(* IEC 61131-3 sources: SJ_AGV/PLC/Standard_functions.4.4.0/CarrierControl, 6 files *)

(* ---- AutoInsert_FB.ST ---- *)
FUNCTION_BLOCK AutoInsert_FB
VAR_EXTERNAL
	NDC8 : NDC8_T;
	INPUT : INPUT_T;

END_VAR

VAR_INPUT

END_VAR

VAR_OUTPUT
		InProgress : BOOL;
		NotInsideTargetSafety : BOOL;
		Failed : BOOL;

END_VAR

VAR

END_VAR
(*************************************************************************************
 		Automatic insert of vehicle into system
**************************************************************************************)

(**************************************************************************************)
(* Make readable/understandable signals

	OUTPUTS	*)
InProgress				:= (NDC8.Autoinsert.Target>0) and not NDC8.LayoutPosition.InSystem;
NotInsideTargetSafety 	:= InProgress and not NDC8.Autoinsert.OnSegment;
Failed					:= (InProgress and NDC8.Guidance.OutsideSafetyZone)
														   or
														   (
																NDC8.Opt.VehicleStatusID = 5
																or NDC8.Opt.VehicleStatusID = 11
														   );

case NDC8.VehicleControl.OperationMode of
	0: 												(* In automatic mode 							*)
		if INPUT.Reset_PB then		(* if reset button pressed 						*)
			NDC8.Manual.PlcSpeed := 50;			(* Set autoinsert speed to 100mm/s 				*)
		else
			NDC8.Manual.PlcSpeed := 0;
		end_if;

	2:
		if ndc8.mcd.Button4 and ndc8.mcd.Button5 then	(* forward slow *)
			ndc8.manual.PlcSpeed := 300 ;
		else
			ndc8.manual.PlcSpeed := 0 ;
		end_if;
else
	;												(* Don't override MCD in semi mode. 			*)
end_case;

END_FUNCTION_BLOCK

(* ---- CARRIERCONTROL_FB.ST ---- *)
FUNCTION_BLOCK CARRIERCONTROL_FB
VAR_EXTERNAL
	(** IN **)
	NDC8 : NDC8_T;

END_VAR

VAR_INPUT
	FlexSlowdown,
	LS2000Slowdown	: bool;
END_VAR

VAR_OUTPUT
	AutoInsertNotInsideTargetSafety : bool;
	AutoinsertInProgress			: bool;
	StartDelayStartWarning			: bool;
END_VAR

VAR

	AutoInsert : AutoInsert_FB;
	SlowDown : Slowdown_FB;
	StartDelay : StartDelay_FB;
	EStopFB : EStop_FB;
	ResetButtonFB : ResetButton_FB;

	MasterLink_TOF	: TOF;

	MasterLinkUp_RT,
	BbxDone_RT,
	NDC8LibFail_RT,
	StandardFBFail_RT		: R_Trig;

	MasterLink_FT		: F_Trig;

	to_bytes : NDC8_STRING_TO_BYTES;
	to_dec : ASCII_TO_DEC;
	AccessPointB5,
	AccessPointB6,
	AccessPointB5b1A,
	AccessPointB5b2A,
	AccessPointB6b1A,
	AccessPointB6b2A,
	AccessPointB5b1,
	AccessPointB6b1,
	AccessPointB5b2,
	AccessPointB6b2,
	MasterLink		 : dint;
	NDC8LibFail,
	StandardFBFail : bool;

	BlackboxFB : Blackbox_FB;

END_VAR
(*
------------------------------------------------------------------------------------
 CARRIER_CONTROL_FB
 ------------------

 Description:
 Handles symbols essential for driving the vehicle
 -------------------------------------------------------------------------------------*)

(**************************************************************************************)

AutoInsert();
Slowdown(	FlexSlowdown := FlexSlowdown,
			LS2000Slowdown := LS2000Slowdown); 			(* Slow down vehicle *)
StartDelay();			(* Start delay after estop *)
EStopFB();
ResetButtonFB();

(**************************************************************************************)

(* Version verification  *)

(**************************************************************************************)
(* ALTRENATIVE CREEP DISTANCE  *)
if NDC8.UserDefined.NormalCreepDistance = 0 then
	NDC8.UserDefined.NormalCreepDistance := NDC8.Vehicle.CreepDistance;
end_if;

(**************************************************************************************)
(* Do not allow download from Application Designer while vehicle is moving *)
NDC8.VehicleControl.PreventAppDownload := NDC8.VehicleControl.Moving;

(**************************************************************************************)
(* Events 		 *)

(* Convert Access points MAC adress xx.xx.xx.xx.b1.b2 from ASCII to dint *)

to_bytes(str:= NDC8.Wlan.AccessPoint);					(* Converts string to bytes *)
AccessPointB5b1A := byte_to_dint(to_bytes.bytes[13]);
AccessPointB5b2A := byte_to_dint(to_bytes.bytes[14]);
AccessPointB6b1A := byte_to_dint(to_bytes.bytes[16]);
AccessPointB6b2A := byte_to_dint(to_bytes.bytes[17]);

to_dec(ASCII:= AccessPointB5b1A);						(* Convert from ASCII to decimal *)
AccessPointB5b1  := to_dec.dec;
to_dec(ASCII:= AccessPointB5b2A);
AccessPointB5b2  := to_dec.dec;
to_dec(ASCII:= AccessPointB6b1A);
AccessPointB6b1  := to_dec.dec;
to_dec(ASCII:= AccessPointB6b2A);
AccessPointB6b2  := to_dec.dec;

MasterLink_TOF(IN:=NDC8.Master.MasterLinkUp, PT:=t#10s);(* Connection is down for more than 10 seconds. *)
MasterLink_FT(CLK:= MasterLink_TOF.q); 					(* Only generate event when connection is lost, not during boot. *)
Case MasterLink of
	0: 	if NDC8.Master.MasterLinkUp then
		(* Found connection to system manager. *)
			MasterLink := 10;
		end_if;
	10: if MasterLink_FT.q then									(* Lost connection to system manager. *)
		BbxTrig := (NDC8.VehicleControl.OperationMode=0);		(* Create blackbox if vehicle is in Automatic Mode. *)
		a:=TRACE_bool('BbxTrig',BbxTrig);
		a:=TRACE_string('MasterLink down');
		NDC8.Blackbox.TrigReason:='MasterLink down';
		MasterLink := 0;
	end_if;
end_case;

(**************************************************************************************)
(* Stop while master controller is minimizes the segments allocated, during detouring. TS40 in NDC demo. *)

if NDC8.VehicleControl.HaltRequest and not StopHalt then
    StopHalt:= True;
    NDC8.VehicleControl.HaltRequestDone:=True;
elsif not NDC8.VehicleControl.HaltRequest and StopHalt then
    NDC8.VehicleControl.HaltRequestDone:=False;
    StopHalt:= False;
end_if;

(* G5 CHECK BATTERY OVER VOLTAGE *)

(**************************************************************************************)
(* 			DEBUG handling *)

if BbxTrig then
	BlackboxFB();
end_if;

BbxDone_RT(CLK:=BlackboxFB.finished);
if BbxDone_RT.q then
	BbxTrig := false;
	a:=TRACE_bool('BbxTrig',BbxTrig);
	NDC8.Blackbox.TrigReason:='Default';
end_if;

(**************************************************************************************)
(* 			Outputs *)
AutoinsertInProgress			:= Autoinsert.InProgress;
AutoInsertNotInsideTargetSafety := AutoInsert.NotInsideTargetSafety;
StartDelayStartWarning			:= StartDelay.StartWarning;

END_FUNCTION_BLOCK

(* ---- ESTOP_FB.ST ---- *)
FUNCTION_BLOCK ESTOP_FB
VAR_EXTERNAL
	NDC8 : NDC8_T;
	INPUT : INPUT_T;
END_VAR

VAR_INPUT

END_VAR

VAR_OUTPUT

END_VAR

VAR
	EstopRT		 	: R_trig;
	EstopFT		 	: R_trig;
	EstopPBRT	 	: R_trig;
END_VAR
(**************************************************************************************)
(* E-STOP BUTTONS: *)

StopEstopButton := INPUT.EstopStop_PB and NDC8.VehicleControl.OperationMode <> 1;	(* Estop push button in all modes except manual *)
StopReset		:= StopReset OR StopEstopButton;									(* This stop signal needs to be reset	*)

(* Display Vehicle E-Stopped *)
DisplayStopString(INStatus:=StopEstopButton, StopString:=8, StopValue:=0);

(* Event  Estop pushbutton ON *)
EStopPBRT(CLK:=StopEstopButton);
if EStopPBRT.Q then
	;
end_if;

(* Event  Estop ON * )

EStopRT(CLK:=NDC8.VehicleControl.Estop);
EStopFT(CLK:=NDC8.VehicleControl.Estop);
if EStopRT.Q then
	EventQueue(EventCode:=100,
			Par1:=NDC8.LayoutPosition.Segment,
			Par2:=0,
			Par3:=0,
			Par4:=0);
	a:=TRACE_DINT('EventCode', EventQueue.EventCode);
end_if;
*)

END_FUNCTION_BLOCK

(* ---- RESETBUTTON_FB.ST ---- *)
FUNCTION_BLOCK RESETBUTTON_FB
VAR_EXTERNAL
	NDC8 : NDC8_T;
	INPUT : INPUT_T;

END_VAR

VAR_INPUT

END_VAR

VAR_OUTPUT

END_VAR

VAR
	StopResetRT,
	ResetButtonRT 	 : r_trig;
	EstopFT,
	ResetButtonFT	 : F_Trig;

END_VAR
(**************************************************************************************)
(* RESET STOP: *)
StopResetRT(CLK:=StopReset);
ResetButtonRT(CLK:=Input.Reset_PB);
ResetButtonFT(CLK:=Input.Reset_PB);

(* Reset push needed *)
if ResetButtonRT.Q and NDC8.LayoutPosition.InSystem then 			(* Set stop signal while button is pressed,
																	so the vehicle does not start to drive,
																	except during autoinsert or during override of rear obstacle *)
	StopResetButton := true;
end_if;

if Input.Reset_PB
	or Input.TillerArmDown
	or Input.GateOpen
	or Input.PlatformNotUpperPos then												(* Release StopReset bit when pressing the button *)
		StopReset 	:= false;
end_if;

if ResetButtonFT.Q or
	NDC8.VehicleControl.OperationMode = 1 then
		StopReset 						:= false;
		StopResetButton 				:= false;
end_if;

InStatus	:= 	StopReset and NDC8.VehicleControl.OperationMode <> 0;
DisplayStopString(INStatus:=InStatus, StopString:=74, StopValue:=0);

InStatus	:= 	StopResetButton	and NDC8.VehicleControl.OperationMode <> 0;
DisplayStopString(INStatus:=InStatus, StopString:=124, StopValue:=0);

END_FUNCTION_BLOCK

(* ---- SLOWDOWN_FB.ST ---- *)
FUNCTION_BLOCK SLOWDOWN_FB
VAR_EXTERNAL
	NDC8 : NDC8_T;
	INPUT : INPUT_T;

END_VAR

VAR_INPUT
	FlexSlowdown,
	LS2000Slowdown	: bool;
END_VAR

VAR_OUTPUT

END_VAR

VAR
	CurrentVehicleSpeed : DINT;
	VehicleSlowDownSpeed : DINT;
	SlowDownTOF : TOF;
	SlowDownKeep : BOOL;
END_VAR
(*************************************************************************************
 		SLOW DOWN
**************************************************************************************)
CurrentVehicleSpeed := abs(NDC8.VehicleControl.SetSpeed);

CurrentVehicleSpeed := CurrentVehicleSpeed / 2;

if CurrentVehicleSpeed < 100 then
	CurrentVehicleSpeed := 100;
end_if;

if FlexSlowDown then									(* Load handling, when entering a pallet *)
	NDC8.VehicleControl.SlowDownSpeed	:= 150;
elsif LS2000Slowdown  then
	NDC8.VehicleControl.SlowDownSpeed:= CurrentVehicleSpeed;
elsif INPUT.SafetyScannerSlowDown then					(* When SlowDown input is set, ramp down in steps *)
	NDC8.VehicleControl.SlowDownSpeed:= CurrentVehicleSpeed;
else
	NDC8.VehicleControl.SlowDownSpeed:= CurrentVehicleSpeed;			(*  speed is 290 to give room for a little variation of current speed,
																		to avoid going over 300 mm/s. *)
end_if;

(* Keep Slowdown bit a little while, after the slow down is released. *)
SlowDownKeep := (INPUT.SafetyScannerSlowDown
					or FlexSlowDown 										(* Load handling, when entering a pallet *)
					or LS2000Slowdown
					or StopReset)											(* Slow start after reset stop *)
				and NDC8.UserDefined.SlowDownDisable <> 2;				(* And SlowDown not disabled from user terminal/display. *)

SlowDownTOF(IN := SlowDownKeep, Pt := t#3s);
NDC8.VehicleControl.SlowDown := SlowDownTOF.Q;

(* Generate events here for System Statistics KPI, to find places with frequent slow downs. *)

END_FUNCTION_BLOCK

(* ---- StartDelay_FB.ST ---- *)
FUNCTION_BLOCK StartDelay_FB
VAR_EXTERNAL
	NDC8 : NDC8_T;
END_VAR

VAR_INPUT
END_VAR

VAR_OUTPUT
	StartWarning : BOOL;
	StartDelayState : DINT;
END_VAR

VAR
	StartDelayShortTOF,
	StartDelayWarningTOF,
	StartDelayLongTOF 		: TOF;
	StartDelayWarningOn,
	StartDelayInactivity,
	StartDelayShort,
	StartDelay,
	StartDelayLong 			: BOOL;
	StartDelayInactivityTON : TON;

END_VAR
(****************************************************************************************)
(* START DELAY  - hold the vehicle for a little while before starting to drive. 		*)

StartDelayInactivity	:= 	NDC8.VehicleControl.OperationMode = 0		(* If standing still on a home position. *)
							and not NDC8.Automatic.ExecDriveCommand
							and not NDC8.Vehicle.Blocked;

StartDelayShortTOF(IN:=StartDelayInactivity, PT:=t#2s);
StartDelayInactivityTON(IN:=StartDelayInactivity, PT:=t#15s);

if NDC8.VehicleControl.OperationMode > 0 then							(* If not ín automatic mode, then start over. *)
	StartDelayState := 0;
end_if;

case StartDelayState of
0: 	(* When stand still on the home for more than 15 seconds. *)
	StopStartDelay 	:= false;
	if StartDelayInactivityTON.q then
		StartDelayState := 10;
		StopStartDelay 	:= true;
	end_if;

10: if not StartDelayInactivity then		(* Wait for a new order. *)
		StartWarning 	:= true;
		StartDelayState := 20;
	end_if;

20: 	(* Hold the vehicle, and beep, for two seconds before starting to drive. *)
	if not StartDelayShortTOF.Q then								(* Stop bit set while on the home station and during the delay. *)
		StartWarning 	:= false;
		StopStartDelay 	:= false;
		StartDelayState := 0;
	end_if;

end_case;

(* Indicate start delay is active when a drive command is recieved. *)
DisplayStopString(INStatus:=StartWarning, StopString:=93, StopValue:=0);
END_FUNCTION_BLOCK
